Staubli VAL3: IOInterface.dtx

public bool bBasicIO1
public bool bBasicIO2
dio diBasicIn[16]
  [0] = {link=BasicIO-1\%I0}
  [1] = {link=BasicIO-1\%I1}
  [2] = {link=BasicIO-1\%I2}
  [3] = {link=BasicIO-1\%I3}
  [4] = {link=BasicIO-1\%I4}
  [5] = {link=BasicIO-1\%I5}
  [6] = {link=BasicIO-1\%I6}
  [7] = {link=BasicIO-1\%I7}
  [8] = {link=BasicIO-1\%I8}
  [9] = {link=BasicIO-1\%I9}
  [10] = {link=BasicIO-1\%I10}
  [11] = {link=BasicIO-1\%I11}
  [12] = {link=BasicIO-1\%I12}
  [13] = {link=BasicIO-1\%I13}
  [14] = {link=BasicIO-1\%I14}
  [15] = {link=BasicIO-1\%I15}
dio diBasicIn2[16]
  [0] = {link=BasicIO-2\%I0}
  [1] = {link=BasicIO-2\%I1}
  [2] = {link=BasicIO-2\%I2}
  [3] = {link=BasicIO-2\%I3}
  [4] = {link=BasicIO-2\%I4}
  [5] = {link=BasicIO-2\%I5}
  [6] = {link=BasicIO-2\%I6}
  [7] = {link=BasicIO-2\%I7}
  [8] = {link=BasicIO-2\%I8}
  [9] = {link=BasicIO-2\%I9}
  [10] = {link=BasicIO-2\%I10}
  [11] = {link=BasicIO-2\%I11}
  [12] = {link=BasicIO-2\%I12}
  [13] = {link=BasicIO-2\%I13}
  [14] = {link=BasicIO-2\%I14}
  [15] = {link=BasicIO-2\%I15}
dio diBasicOut[16]
  [0] = {link=FastIO\fOut0}
  [1] = {link=FastIO\fOut1}
  [2] = {link=BasicIO-1\%Q2}
  [3] = {link=BasicIO-1\%Q3}
  [4] = {link=BasicIO-1\%Q4}
  [5] = {link=BasicIO-1\%Q5}
  [6] = {link=BasicIO-1\%Q6}
  [7] = {link=BasicIO-1\%Q7}
  [8] = {link=BasicIO-1\%Q8}
  [9] = {link=BasicIO-1\%Q9}
  [10] = {link=BasicIO-1\%Q10}
  [11] = {link=BasicIO-1\%Q11}
  [12] = {link=BasicIO-1\%Q12}
  [13] = {link=BasicIO-1\%Q13}
  [14] = {link=BasicIO-1\%Q14}
  [15] = {link=BasicIO-1\%Q15}
dio diBasicOut2[16]
  [0] = {link=BasicIO-2\%Q0}
  [1] = {link=BasicIO-2\%Q1}
  [2] = {link=BasicIO-2\%Q2}
  [3] = {link=BasicIO-2\%Q3}
  [4] = {link=BasicIO-2\%Q4}
  [5] = {link=BasicIO-2\%Q5}
  [6] = {link=BasicIO-2\%Q6}
  [7] = {link=BasicIO-2\%Q7}
  [8] = {link=BasicIO-2\%Q8}
  [9] = {link=BasicIO-2\%Q9}
  [10] = {link=BasicIO-2\%Q10}
  [11] = {link=BasicIO-2\%Q11}
  [12] = {link=BasicIO-2\%Q12}
  [13] = {link=BasicIO-2\%Q13}
  [14] = {link=BasicIO-2\%Q14}
  [15] = {link=BasicIO-2\%Q15}
dio diUserIn[2]
  [0] = {link=usrIn0}
  [1] = {link=usrIn1}
dio diValveOut[2]
  [0] = {link=ValveIO\valve1}
  [1] = {link=ValveIO\valve2}
